ABB RobotStudio station: ABB robot domino project.rspag

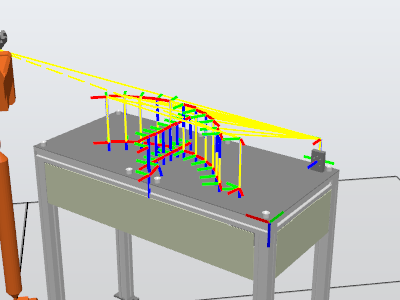
--- station ---
Station lab04_robot_mic (saved by RobotStudio 23.4.10609.1)
Controller R1400
  mechanical unit ROB_1: IRB1400_5_144__01, 6 joints, base frame (0, 0, 0) mm
Layout (positions relative to the parent item):
  - IRB1400_5_144__01 [mechanism, from Robots\IRB1400_5_144__01.rslib] at (0, 0, 0) mm; joint values [0, 0, 0, 0, 0.5236, 0] (rad or m)
  - Stoc1400 [smart component, from Components\Stoc1400.rslib] at (629.33, -613.77, 0) mm, rotated rx 0 ry 0 rz -45 deg
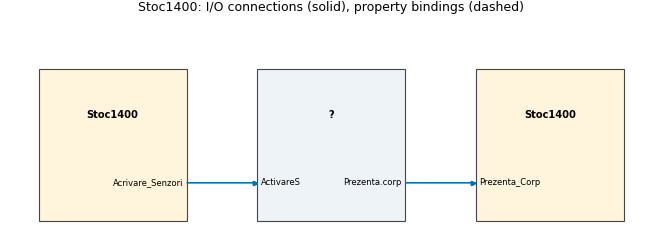
      connections:
        Stoc1400.Acrivare_Senzori -> ?.ActivareS
        Stoc1400.Acrivare_Senzori -> ?.ActivareS
        ?.Prezenta.corp -> Stoc1400.Prezenta_Corp
        ?.Prezenta.corp -> Stoc1400.Prezenta_Corp
    - 679#Body 1 [part, from Components\Stoc1400.rslib]
    - 681#Body 2 [part, from Components\Stoc1400.rslib]
    - 683#Body 3 [part, from Components\Stoc1400.rslib]
    - 685#Body 4 [part, from Components\Stoc1400.rslib]
    - 687#Body 5 [part, from Components\Stoc1400.rslib]
    - 689#Body 6 [part, from Components\Stoc1400.rslib]
    - 691#Body 7 [part, from Components\Stoc1400.rslib]
    - 693#Body 8 [part, from Components\Stoc1400.rslib]
    - 695#Body 9 [part, from Components\Stoc1400.rslib]
    - 697#Body 10 [part, from Components\Stoc1400.rslib]
    - 701#Body 12 [part, from Components\Stoc1400.rslib]
    - 703#Body 13 [part, from Components\Stoc1400.rslib]
    - 705#Body 14 [part, from Components\Stoc1400.rslib]
    - 707#Body 15 [part, from Components\Stoc1400.rslib]
    - 755#Body 39 [part, from Components\Stoc1400.rslib]
    - 757#Body 40 [part, from Components\Stoc1400.rslib]
    - 759#Body 41 [part, from Components\Stoc1400.rslib]
    - 761#Body 42 [part, from Components\Stoc1400.rslib]
    - 785#Body 54 [part, from Components\Stoc1400.rslib]
    - 787#Body 55 [part, from Components\Stoc1400.rslib]
    - 789#Body 56 [part, from Components\Stoc1400.rslib]
    - 791#Body 57 [part, from Components\Stoc1400.rslib]
    - 793#Body 58 [part, from Components\Stoc1400.rslib]
    - Part [part, from Components\Stoc1400.rslib]
    - Part_2 [part, from Components\Stoc1400.rslib]
    - Part_3 [part, from Components\Stoc1400.rslib]
    - Part_4 [part, from Components\Stoc1400.rslib]
  - Gripper_R1400 [smart component] at (943.61, 0, 1152.5) mm, rotated rx 180 ry 60 rz 180 deg
      signals: DI Open, DO Opened
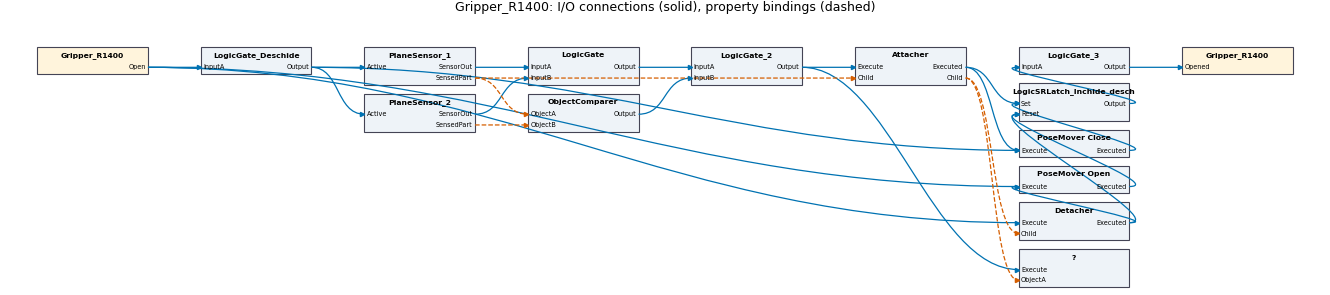
      connections:
        Attacher.Executed -> LogicSRLatch_Inchide_deschide.Set
        Detacher.Executed -> LogicSRLatch_Inchide_deschide.Reset
        Attacher.Executed -> PoseMover Close.Execute
        PoseMover Close.Executed -> LogicSRLatch_Inchide_deschide.Set
        Detacher.Executed -> PoseMover Open.Execute
        PoseMover Open.Executed -> LogicSRLatch_Inchide_deschide.Reset
        LogicGate.Output -> LogicGate_2.InputA
        ObjectComparer.Output -> LogicGate_2.InputB
        LogicGate_2.Output -> ?.Execute
        LogicGate_2.Output -> Attacher.Execute
        PlaneSensor_1.SensorOut -> LogicGate.InputA
        PlaneSensor_2.SensorOut -> LogicGate.InputB
        LogicGate_Deschide.Output -> PlaneSensor_2.Active
        LogicGate_Deschide.Output -> PlaneSensor_1.Active
        LogicGate_Deschide.Output -> PoseMover Close.Execute
        LogicSRLatch_Inchide_deschide.Output -> LogicGate_3.InputA
        LogicGate_3.Output -> Gripper_R1400.Opened
        Gripper_R1400.Open -> LogicGate_Deschide.InputA
        Gripper_R1400.Open -> Detacher.Execute
        Gripper_R1400.Open -> PoseMover Open.Execute
        Attacher.Child => Detacher.Child
        Attacher.Child => ?.ObjectA
        PlaneSensor_1.SensedPart => Attacher.Child
        PlaneSensor_1.SensedPart => ObjectComparer.ObjectA
        PlaneSensor_2.SensedPart => ObjectComparer.ObjectB
    - Attacher [smart component]
        properties: Parent=Gripper; Flange=0; Child=(none); Mount=false; Offset=[0 0 0]; Orientation=[0 0 0]
        signals: DI Execute, DO Executed
    - Detacher [smart component]
        properties: Child=(none); KeepPosition=true
        signals: DI Execute, DO Executed
    - LogicGate_Deschide [smart component]
        properties: Operator=NOT; Delay=0
        signals: DI InputA, DI InputB, DO Output
    - LogicSRLatch_Inchide_deschide [smart component]
        signals: DI Set, DI Reset, DO Output, DO InvOutput
    - PoseMover Close [smart component]
        properties: Mechanism=Gripper; Pose=3; Duration=0
        signals: DI Execute, DI Pause, DI Cancel, DO Executed, DO Executing, DO Paused
    - PoseMover Open [smart component]
        properties: Mechanism=Gripper; Pose=2; Duration=0
        signals: DI Execute, DI Pause, DI Cancel, DO Executed, DO Executing, DO Paused
    - ObjectComparer [smart component, from Components\ObjectComparer.rslib]
        properties: ObjectA=(none); ObjectB=(none)
    - LogicGate [smart component, from Components\LogicGate.rslib]
        properties: Operator=AND; Delay=0
    - LogicGate_2 [smart component, from Components\LogicGate.rslib]
        properties: Operator=AND; Delay=0
    - PlaneSensor_1 [smart component, from Components\PlaneSensor.rslib]
        properties: Origin=[-0.015 0.017 0.128]; Axis1=[2.03942606365875E-08 6.36094387840794E-09 0.0549999999999959]; Axis2=[0.03 0 0]; SensedPart=(none); Tag=(none)
      - _sensorPart_ [part], size 30 x 0 x 55 mm
    - PlaneSensor_2 [smart component, from Components\PlaneSensor.rslib]
        properties: Origin=[-0.015 -0.017 0.128]; Axis1=[0 0 0.055]; Axis2=[0.03 0 0]; SensedPart=(none); Tag=(none)
      - _sensorPart_ [part], size 30 x 0 x 55 mm
    - Gripper [mechanism] at (0, 0.03, 0) mm; joint values [0, 0] (rad or m)
        TCP Efector at (0, 0, 184.3) mm
        links: L1, L2, L3
    - LogicGate_3 [smart component, from Components\LogicGate.rslib]
        properties: Operator=NOT; Delay=0
  - Piesa_A [part, from Components\Piesa_A.rslib] at (465.74, -1014.9, 834) mm, rotated rx 84.55 ry 90 rz -140.46 deg
  - Piesa_C [part, from Components\Piesa_C.rslib] at (465.74, -1014.9, 834) mm, rotated rx 84.55 ry 90 rz -140.46 deg
  - Piesa_D [part, from Components\Piesa_D.rslib] at (465.74, -1014.9, 834) mm, rotated rx 84.55 ry 90 rz -140.46 deg
  - Piesa_C_2 [part, from Components\Piesa_C.rslib] at (465.74, -1014.9, 834) mm, rotated rx 84.55 ry 90 rz -140.46 deg
  - Piesa_C_3 [part, from Components\Piesa_C2.rslib] at (465.74, -1014.9, 834) mm, rotated rx 84.55 ry 90 rz -140.46 deg
  - Piesa_C_4 [part, from Components\Piesa_C2.rslib] at (465.74, -1014.9, 834) mm, rotated rx 84.55 ry 90 rz -140.46 deg
  - Piesa_C_5 [part, from Components\Piesa_C2.rslib] at (465.74, -1014.9, 834) mm, rotated rx 84.55 ry 90 rz -140.46 deg
  - Piesa [part, from Components\Piesa_D.rslib] at (465.74, -1014.9, 834) mm, rotated rx 84.55 ry 90 rz -140.46 deg
  - Piesa_D_2 [part, from Components\Piesa_D_1.rslib] at (465.74, -1014.9, 834) mm, rotated rx 84.55 ry 90 rz -140.46 deg
  - Piesa_E [part, from Components\Piesa_E.rslib] at (465.74, -1014.9, 834) mm, rotated rx 84.55 ry 90 rz -140.46 deg
  - Piesa_F [part, from Components\Piesa_F.rslib] at (465.74, -1014.9, 834) mm, rotated rx 84.55 ry 90 rz -140.46 deg
  - Piesa_A_2 [part, from Components\Piesa_A2.rslib] at (465.74, -1014.9, 834) mm, rotated rx 84.55 ry 90 rz -140.46 deg
  - Piesa_A_3 [part, from Components\Piesa_A3.rslib] at (465.74, -1014.9, 834) mm, rotated rx 84.55 ry 90 rz -140.46 deg
  - Piesa_A_4 [part, from Components\Piesa_A4.rslib] at (465.74, -1014.9, 834) mm, rotated rx 84.55 ry 90 rz -140.46 deg
Attachment: Gripper_R1400 is attached to IRB1400_5_144__01 / Link6
Station logic (signal -> signal, property => property):
  R1400.DO10_9 -> Gripper_R1400.Open
Targets, tools, work objects and paths stored in the station and not in the controller backup, written as RAPID:
! task T_ROB1
MODULE Module1
  CONST robtarget aPiesa:=[[50.700017393,375.465881391,-34],[0.499999623,0.499998418,-0.500001769,0.50000019],[-1,0,-1,0],[9E+09,9E+09,9E+09,9E+09,9E+09,9E+09]];
ENDMODULE


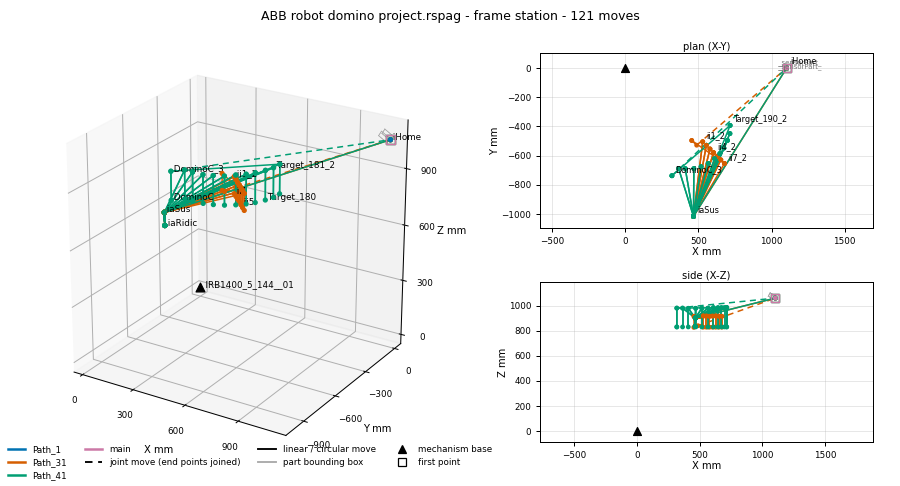
[picture p0: tool path of ABB robot domino project.rspag in frame station, 121 of 121 moves have a stored position in this frame; points joined in program order, loops and branches not executed]
--- Controller Data/R1400/RAPID/TASK1/PROGMOD/CalibData.mod ---
MODULE CalibData
ENDMODULE

--- Controller Data/R1400/RAPID/TASK1/PROGMOD/Module1.mod ---
MODULE Module1
    LOCAL PERS tooldata Efector:=[TRUE,[[0,0.033033672,184.3],[1,0,0,0]],[1.5,[0,0,90],[1,0,0,0],0.01,0.01,0.01]];
    LOCAL PERS wobjdata Paleta:=[FALSE,TRUE,"",[[164.402459193,-785.24154085,800],[0,0.923888632,0.382661463,0]],[[0,0,0],[1,0,0,0]]];
    LOCAL CONST robtarget Target_10:=[[50.700017393,375.465881391,-34],[0.69868606,0.000100025,0.000759531,-0.715427986],[0,0,0,0],[9E+09,9E+09,9E+09,9E+09,9E+09,9E+09]];
    CONST robtarget Target_20:=[[456.326,269.195,-115.604996843],[0.698683796,0.000101541,0.000757843,-0.715430199],[-1,0,-1,0],[9E+09,9E+09,9E+09,9E+09,9E+09,9E+09]];
    CONST robtarget iHome:=[[1219.122841698,108.513746508,-260.35],[0.331394548,-0.461944316,-0.191330732,-0.800111026],[0,-1,0,0],[9E+09,9E+09,9E+09,9E+09,9E+09,9E+09]];
    CONST robtarget iaSus:=[[50.700017393,375.465881391,-101.41254067],[0.707106781,0,0,-0.707106781],[-1,0,-1,0],[9E+09,9E+09,9E+09,9E+09,9E+09,9E+09]];
    CONST robtarget iaRidic:=[[52.292573517,372.97750672,-34],[0.69868606,0.000100025,0.000759531,-0.715427986],[-1,0,-1,0],[9E+09,9E+09,9E+09,9E+09,9E+09,9E+09]];
    CONST robtarget ii1_2:=[[456.326,59.195,-118.568809292],[0.698683796,0.000101541,0.000757843,-0.715430199],[0,0,0,0],[9E+09,9E+09,9E+09,9E+09,9E+09,9E+09]];
    CONST robtarget ii1:=[[456.326,59.195,-28.603],[0.698683796,0.000101541,0.000757843,-0.715430199],[0,0,0,0],[9E+09,9E+09,9E+09,9E+09,9E+09,9E+09]];
    CONST robtarget ii2_2:=[[456.326,94.195,-117.638928881],[0.698683796,0.000101541,0.000757843,-0.715430199],[0,0,0,0],[9E+09,9E+09,9E+09,9E+09,9E+09,9E+09]];
    CONST robtarget ii2:=[[456.326,94.195,-28.603],[0.698683796,0.000101541,0.000757843,-0.715430199],[0,0,0,0],[9E+09,9E+09,9E+09,9E+09,9E+09,9E+09]];
    CONST robtarget ii3_2:=[[456.326,129.195,-115.401644855],[0.698683796,0.000101541,0.000757843,-0.715430199],[0,0,0,0],[9E+09,9E+09,9E+09,9E+09,9E+09,9E+09]];
    CONST robtarget ii3:=[[456.326,129.195,-28.603],[0.698683796,0.000101541,0.000757843,-0.715430199],[0,0,0,0],[9E+09,9E+09,9E+09,9E+09,9E+09,9E+09]];
    CONST robtarget ii4_2:=[[456.326,164.195,-116.998692265],[0.698683796,0.000101541,0.000757843,-0.715430199],[0,0,0,0],[9E+09,9E+09,9E+09,9E+09,9E+09,9E+09]];
    CONST robtarget ii4:=[[456.326,164.195,-28.603],[0.698683796,0.000101541,0.000757843,-0.715430199],[0,0,0,0],[9E+09,9E+09,9E+09,9E+09,9E+09,9E+09]];
    CONST robtarget ii5_2:=[[456.326,199.195,-117.832130834],[0.698683796,0.000101541,0.000757843,-0.715430199],[0,0,0,0],[9E+09,9E+09,9E+09,9E+09,9E+09,9E+09]];
    CONST robtarget ii5:=[[456.326,199.195,-28.603],[0.698683796,0.000101541,0.000757843,-0.715430199],[0,0,0,0],[9E+09,9E+09,9E+09,9E+09,9E+09,9E+09]];
    CONST robtarget ii6_2:=[[456.326,234.195,-116.561054339],[0.698683796,0.000101541,0.000757843,-0.715430199],[0,0,0,0],[9E+09,9E+09,9E+09,9E+09,9E+09,9E+09]];
    CONST robtarget ii6:=[[456.326,234.195,-28.603],[0.698683796,0.000101541,0.000757843,-0.715430199],[0,0,0,0],[9E+09,9E+09,9E+09,9E+09,9E+09,9E+09]];
    CONST robtarget ii7_2:=[[456.326,269.195,-115.604996843],[0.698683796,0.000101541,0.000757843,-0.715430199],[0,0,0,0],[9E+09,9E+09,9E+09,9E+09,9E+09,9E+09]];
    CONST robtarget ii7:=[[456.326,269.195,-28.603],[0.698683796,0.000101541,0.000757843,-0.715430199],[0,0,0,0],[9E+09,9E+09,9E+09,9E+09,9E+09,9E+09]];
    CONST robtarget ID_Sus:=[[409.258836726,-0.15273945,-115.604996843],[0.698683796,0.000101541,0.000757843,-0.715430199],[-1,0,-1,0],[9E+09,9E+09,9E+09,9E+09,9E+09,9E+09]];
    CONST robtarget ID_Jos:=[[409.258836726,-0.15273945,-26.947996726],[0.698683796,0.000101541,0.000757843,-0.715430199],[-1,0,-1,0],[9E+09,9E+09,9E+09,9E+09,9E+09,9E+09]];
    CONST robtarget Domino:=[[410.25163548,46.685138582,-40.418213822],[0.68917084,-0.113675498,-0.121440524,-0.705247214],[-1,0,-1,0],[9E+09,9E+09,9E+09,9E+09,9E+09,9E+09]];
    CONST robtarget Target_170_2:=[[481.800724938,199.544231585,-183.999604819],[0.995072185,0,0,-0.099153148],[-1,0,0,0],[9E+09,9E+09,9E+09,9E+09,9E+09,9E+09]];
    CONST robtarget Target_170:=[[481.800724938,199.544231585,-30.630486906],[0.995072185,0,0,-0.099153148],[0,0,0,0],[9E+09,9E+09,9E+09,9E+09,9E+09,9E+09]];
    CONST robtarget Target_180_2:=[[582.438198055,172.573372066,-183.959345103],[0.97629086,0,0,-0.216462829],[-1,-1,0,0],[9E+09,9E+09,9E+09,9E+09,9E+09,9E+09]];
    CONST robtarget Target_180:=[[582.438198055,172.573372066,-30.630486906],[0.97629086,0,0,-0.216462829],[0,0,0,0],[9E+09,9E+09,9E+09,9E+09,9E+09,9E+09]];
    CONST robtarget Target_190_2:=[[667.781911679,112.809011422,-184.493963186],[0.923870432,0,0,-0.382705401],[0,0,0,0],[9E+09,9E+09,9E+09,9E+09,9E+09,9E+09]];
    CONST robtarget Target_190:=[[667.781911679,112.809011422,-30.630486906],[0.923870432,0,0,-0.382705401],[0,0,0,0],[9E+09,9E+09,9E+09,9E+09,9E+09,9E+09]];
    CONST robtarget Target_200_2:=[[306.909359491,163.530688918,-167.727227508],[0.536299591,0.000254363,0.000722629,-0.844027347],[-1,0,-1,0],[9E+09,9E+09,9E+09,9E+09,9E+09,9E+09]];
    CONST robtarget Target_200:=[[306.909359491,163.530688918,-26.975190983],[0.536299591,0.000254363,0.000722629,-0.844027347],[-1,0,-1,0],[9E+09,9E+09,9E+09,9E+09,9E+09,9E+09]];
    CONST robtarget Target_210_2:=[[354.733930359,180.209703677,-168.853762894],[0.464361971,0.000313489,0.000699011,-0.885645173],[-1,-1,-1,0],[9E+09,9E+09,9E+09,9E+09,9E+09,9E+09]];
    CONST robtarget Target_210:=[[354.733930359,180.209703677,-26.975190983],[0.464361971,0.000313489,0.000699011,-0.885645173],[-1,-1,-1,0],[9E+09,9E+09,9E+09,9E+09,9E+09,9E+09]];
    CONST robtarget Target_220_2:=[[403.502030206,179.286180207,-166.530198208],[0.375825673,0.00038013,0.000665127,-0.926690065],[-1,-1,-1,0],[9E+09,9E+09,9E+09,9E+09,9E+09,9E+09]];
    CONST robtarget Target_220:=[[403.502030206,179.286180207,-26.975190983],[0.375825673,0.00038013,0.000665127,-0.926690065],[-1,-1,-1,0],[9E+09,9E+09,9E+09,9E+09,9E+09,9E+09]];
    CONST robtarget Target_230_2:=[[451.347703104,167.719972633,-167.069743011],[0.258943654,0.000459083,0.000613298,-0.965892125],[-1,-1,-1,0],[9E+09,9E+09,9E+09,9E+09,9E+09,9E+09]];
    CONST robtarget Target_230:=[[451.347703104,167.719972633,-26.975190983],[0.258943654,0.000459083,0.000613298,-0.965892125],[-1,-1,-1,0],[9E+09,9E+09,9E+09,9E+09,9E+09,9E+09]];
    CONST robtarget DominoC_3:=[[142.859438409,74.577988932,-180.688995332],[0.393881017,0,0,-0.919161435],[-1,0,-1,0],[9E+09,9E+09,9E+09,9E+09,9E+09,9E+09]];
    CONST robtarget DominoC:=[[142.859438409,74.577988932,-30.630486906],[0.393881017,0,0,-0.919161435],[-1,0,-1,0],[9E+09,9E+09,9E+09,9E+09,9E+09,9E+09]];
    CONST robtarget Lovire:=[[241.300943539,67.077354326,-28.34493513],[0.698121404,-0.033467609,-0.042039078,-0.713960182],[-1,0,-1,0],[9E+09,9E+09,9E+09,9E+09,9E+09,9E+09]];
    CONST robtarget Target_150_2:=[[283.578545465,146.440862541,-179.015978792],[0.300007552,-0.00000002,-0.000000178,-0.953936826],[-1,-1,-1,0],[9E+09,9E+09,9E+09,9E+09,9E+09,9E+09]];
    CONST robtarget Target_160:=[[378.007856837,190.468506271,-30.630486906],[0.130502616,0,0,-0.991447965],[-1,-1,-1,0],[9E+09,9E+09,9E+09,9E+09,9E+09,9E+09]];
    CONST robtarget Target_171_2:=[[528.22113049,192.308253683,-184.191222664],[0.984830453,0,0,-0.173519391],[-1,-1,0,0],[9E+09,9E+09,9E+09,9E+09,9E+09,9E+09]];
    CONST robtarget Target_171:=[[528.22113049,192.308253683,-30.630486906],[0.984830453,0,0,-0.173519391],[-1,-1,0,0],[9E+09,9E+09,9E+09,9E+09,9E+09,9E+09]];
    CONST robtarget Target_141:=[[241.884072512,104.750355256,-30.630486906],[0.349991593,0,0,-0.936752841],[-1,0,-1,0],[9E+09,9E+09,9E+09,9E+09,9E+09,9E+09]];
    CONST robtarget Target_140:=[[209.902359402,72.771684008,-30.562172725],[0.393881017,0,0,-0.919161435],[-1,0,-1,0],[9E+09,9E+09,9E+09,9E+09,9E+09,9E+09]];
    CONST robtarget Target_140_2:=[[209.902359402,72.771684008,-180.562172725],[0.393881017,0,0,-0.919161435],[-1,0,-1,0],[9E+09,9E+09,9E+09,9E+09,9E+09,9E+09]];
    CONST robtarget Target_150:=[[283.616805576,146.386732955,-30.630438676],[0.300007552,-0.00000002,-0.000000178,-0.953936826],[-1,-1,-1,0],[9E+09,9E+09,9E+09,9E+09,9E+09,9E+09]];
    CONST robtarget Target_161_2:=[[431.263927092,198.857293079,-184.181538316],[0.021799568,0,0,-0.999762361],[-1,-1,-1,0],[9E+09,9E+09,9E+09,9E+09,9E+09,9E+09]];
    CONST robtarget Target_141_2:=[[241.884072512,104.750355256,-179.064848292],[0.349991593,0,0,-0.936752841],[-1,0,-1,0],[9E+09,9E+09,9E+09,9E+09,9E+09,9E+09]];
    CONST robtarget Target_151_2:=[[327.822781481,171.759911975,-180.139566205],[0.223808464,0,0,-0.974633147],[-1,0,-1,0],[9E+09,9E+09,9E+09,9E+09,9E+09,9E+09]];
    CONST robtarget Target_181:=[[627.363553937,151.187326706,-30.978234387],[0.949049924,0,0,-0.315125754],[-1,-1,0,0],[9E+09,9E+09,9E+09,9E+09,9E+09,9E+09]];
    CONST robtarget Target_151:=[[327.822781481,171.759911975,-30.630486906],[0.223808464,0,0,-0.974633147],[-1,-1,-1,0],[9E+09,9E+09,9E+09,9E+09,9E+09,9E+09]];
    CONST robtarget Target_161:=[[431.263927092,198.857293079,-30.630486906],[0.021799568,0,0,-0.999762361],[-1,-1,-1,0],[9E+09,9E+09,9E+09,9E+09,9E+09,9E+09]];
    CONST robtarget Target_160_2:=[[378.007856837,190.468506271,-180.335566752],[0.130502616,0,0,-0.991447965],[-1,-1,-1,0],[9E+09,9E+09,9E+09,9E+09,9E+09,9E+09]];
    CONST robtarget Target_181_2:=[[627.363553937,151.187326706,-184.978843448],[0.949049924,0,0,-0.315125754],[-1,-1,0,0],[9E+09,9E+09,9E+09,9E+09,9E+09,9E+09]];
    CONST robtarget LovireCerc:=[[142.868157241,74.605504654,-30.630477518],[0.756533746,0.000000012,0.000000022,-0.653954656],[-1,0,-1,0],[9E+09,9E+09,9E+09,9E+09,9E+09,9E+09]];
    LOCAL PROC Path_1()
        MoveJ iHome,v300,fine,Efector\WObj:=Paleta;
    ENDPROC

    LOCAL PROC Path_31()
        Set DO10_9;
        WaitTime 0.5;
        MoveJ iHome,v300,fine,Efector\WObj:=Paleta;
        WaitTime 0.5;
        MoveL iaSus,v300,fine,Efector\WObj:=Paleta;
        WaitTime 0.5;
        MoveL iaRidic,v300,fine,Efector\WObj:=Paleta;
        WaitTime 0.5;
        Reset DO10_9;
        WaitTime 0.5;
        MoveL iaSus,v300,fine,Efector\WObj:=Paleta;
        WaitTime 0.5;
        MoveL ii1_2,v300,fine,Efector\WObj:=Paleta;
        WaitTime 0.5;
        MoveL ii1,v300,fine,Efector\WObj:=Paleta;
        Set DO10_9;
        WaitTime 0.5;
        MoveL ii1_2,v300,fine,Efector\WObj:=Paleta;
        WaitTime 0.5;
        MoveL iaSus,v300,fine,Efector\WObj:=Paleta;
        WaitTime 0.5;
        MoveL iaRidic,v300,fine,Efector\WObj:=Paleta;
        WaitTime 0.5;
        Reset DO10_9;
        WaitTime 0.5;
        MoveL iaSus,v300,fine,Efector\WObj:=Paleta;
        WaitTime 0.5;
        Reset DO10_9;
        WaitTime 0.5;
        MoveL ii2_2,v300,fine,Efector\WObj:=Paleta;
        WaitTime 0.5;
        MoveL ii2,v300,fine,Efector\WObj:=Paleta;
        WaitTime 0.5;
        Set DO10_9;
        WaitTime 0.5;
        MoveL ii2_2,v300,fine,Efector\WObj:=Paleta;
        WaitTime 0.5;
        MoveL iaSus,v300,fine,Efector\WObj:=Paleta;
        WaitTime 0.5;
        MoveL iaRidic,v300,fine,Efector\WObj:=Paleta;
        WaitTime 0.5;
        Reset DO10_9;
        WaitTime 0.5;
        MoveL iaSus,v300,fine,Efector\WObj:=Paleta;
        WaitTime 0.5;
        Reset DO10_9;
        WaitTime 0.5;
        MoveL ii3_2,v300,fine,Efector\WObj:=Paleta;
        WaitTime 0.5;
        MoveL ii3,v300,fine,Efector\WObj:=Paleta;
        WaitTime 0.5;
        Set DO10_9;
        WaitTime 0.5;
        MoveL ii3_2,v300,fine,Efector\WObj:=Paleta;
        WaitTime 0.5;
        MoveL iaSus,v300,fine,Efector\WObj:=Paleta;
        WaitTime 0.5;
        MoveL iaRidic,v300,fine,Efector\WObj:=Paleta;
        WaitTime 0.5;
        Reset DO10_9;
        WaitTime 0.5;
        MoveL iaSus,v300,fine,Efector\WObj:=Paleta;
        WaitTime 0.5;
        Reset DO10_9;
        WaitTime 0.5;
        MoveL ii4_2,v300,fine,Efector\WObj:=Paleta;
        WaitTime 0.5;
        MoveL ii4,v300,fine,Efector\WObj:=Paleta;
        WaitTime 0.5;
        Set DO10_9;
        WaitTime 0.5;
        MoveL ii4_2,v300,fine,Efector\WObj:=Paleta;
        WaitTime 0.5;
        MoveL iaSus,v300,fine,Efector\WObj:=Paleta;
        WaitTime 0.5;
        MoveL iaRidic,v300,fine,Efector\WObj:=Paleta;
        WaitTime 0.5;
        Reset DO10_9;
        MoveL iaSus,v300,fine,Efector\WObj:=Paleta;
        WaitTime 0.5;
        Reset DO10_9;
        WaitTime 0.5;
        MoveL ii5_2,v300,fine,Efector\WObj:=Paleta;
        WaitTime 0.5;
        MoveL ii5,v300,fine,Efector\WObj:=Paleta;
        WaitTime 0.5;
        Set DO10_9;
        WaitTime 0.5;
        MoveL ii5_2,v300,fine,Efector\WObj:=Paleta;
        WaitTime 0.5;
        MoveL iaSus,v300,fine,Efector\WObj:=Paleta;
        WaitTime 0.5;
        MoveL iaRidic,v300,fine,Efector\WObj:=Paleta;
        WaitTime 0.5;
        Reset DO10_9;
        MoveL iaSus,v300,fine,Efector\WObj:=Paleta;
        WaitTime 0.5;
        Reset DO10_9;
        WaitTime 0.5;
        MoveL ii6_2,v300,fine,Efector\WObj:=Paleta;
        WaitTime 0.5;
        MoveL ii6,v300,fine,Efector\WObj:=Paleta;
        WaitTime 0.5;
        Set DO10_9;
        WaitTime 0.5;
        MoveL ii6_2,v300,fine,Efector\WObj:=Paleta;
        WaitTime 0.5;
        MoveL iaSus,v300,fine,Efector\WObj:=Paleta;
        WaitTime 0.5;
        MoveL iaRidic,v300,fine,Efector\WObj:=Paleta;
        WaitTime 0.5;
        WaitTime 0.5;
        Reset DO10_9;
        WaitTime 0.5;
        MoveL iaSus,v300,fine,Efector\WObj:=Paleta;
        WaitTime 0.5;
        Reset DO10_9;
        WaitTime 0.5;
        MoveL ii7_2,v300,fine,Efector\WObj:=Paleta;
        WaitTime 0.5;
        MoveL ii7,v300,fine,Efector\WObj:=Paleta;
        WaitTime 0.5;
        Set DO10_9;
        WaitTime 0.5;
        MoveL ii7_2,v300,fine,Efector\WObj:=Paleta;
        WaitTime 0.5;
        Set DO10_9;
        WaitTime 0.5;
        MoveL ID_Sus,v300,fine,Efector\WObj:=Paleta;
        WaitTime 0.5;
        MoveL ID_Jos,v300,fine,Efector\WObj:=Paleta;
        WaitTime 0.5;
        MoveL Domino,v300,fine,Efector\WObj:=Paleta;
        WaitTime 0.5;
        MoveJ iHome,v300,fine,Efector\WObj:=Paleta;
    ENDPROC

    PROC Path_41()
        Set DO10_9;
        WaitTime 0.5;
        MoveJ iHome,v300,fine,Efector\WObj:=Paleta;
        WaitTime 0.5;
        MoveL iaSus,v300,fine,Efector\WObj:=Paleta;
        WaitTime 0.5;
        MoveL iaRidic,v300,fine,Efector\WObj:=Paleta;
        WaitTime 0.5;
        Reset DO10_9;
        WaitTime 0.5;
        MoveL iaSus,v300,fine,Efector\WObj:=Paleta;
        WaitTime 0.5;
        MoveL Target_140_2,v300,fine,Efector\WObj:=Paleta;
        MoveL Target_140,v300,fine,Efector\WObj:=Paleta;
        WaitTime 0.5;
        Set DO10_9;
        WaitTime 0.5;
        MoveL Target_140_2,v300,fine,Efector\WObj:=Paleta;
        MoveL iaSus,v300,fine,Efector\WObj:=Paleta;
        WaitTime 0.5;
        MoveL iaRidic,v300,fine,Efector\WObj:=Paleta;
        WaitTime 0.5;
        Reset DO10_9;
        WaitTime 0.5;
        MoveL iaSus,v300,fine,Efector\WObj:=Paleta;
        WaitTime 0.5;
        MoveL Target_141_2,v300,fine,Efector\WObj:=Paleta;
        MoveL Target_141,v300,fine,Efector\WObj:=Paleta;
        WaitTime 0.5;
        Set DO10_9;
        WaitTime 0.5;
        MoveL Target_141_2,v300,fine,Efector\WObj:=Paleta;
        MoveL iaSus,v300,fine,Efector\WObj:=Paleta;
        WaitTime 0.5;
        MoveL iaRidic,v300,fine,Efector\WObj:=Paleta;
        WaitTime 0.5;
        Reset DO10_9;
        WaitTime 0.5;
        MoveL iaSus,v300,fine,Efector\WObj:=Paleta;
        WaitTime 0.5;
        MoveL Target_150_2,v300,fine,Efector\WObj:=Paleta;
        MoveL Target_150,v300,fine,Efector\WObj:=Paleta;
        WaitTime 0.5;
        Set DO10_9;
        WaitTime 0.5;
        MoveL Target_150_2,v300,fine,Efector\WObj:=Paleta;
        MoveL iaSus,v300,fine,Efector\WObj:=Paleta;
        WaitTime 0.5;
        MoveL iaRidic,v300,fine,Efector\WObj:=Paleta;
        WaitTime 0.5;
        Reset DO10_9;
        WaitTime 0.5;
        MoveL iaSus,v300,fine,Efector\WObj:=Paleta;
        WaitTime 0.5;
        MoveL Target_151_2,v300,fine,Efector\WObj:=Paleta;
        MoveL Target_151,v300,fine,Efector\WObj:=Paleta;
        WaitTime 0.5;
        Set DO10_9;
        WaitTime 0.5;
        MoveL Target_151_2,v300,fine,Efector\WObj:=Paleta;
        MoveL iaSus,v300,fine,Efector\WObj:=Paleta;
        WaitTime 0.5;
        MoveL iaRidic,v300,fine,Efector\WObj:=Paleta;
        WaitTime 0.5;
        Reset DO10_9;
        WaitTime 0.5;
        MoveL iaSus,v300,fine,Efector\WObj:=Paleta;
        WaitTime 0.5;
        MoveL Target_160_2,v300,fine,Efector\WObj:=Paleta;
        MoveL Target_160,v300,fine,Efector\WObj:=Paleta;
        WaitTime 0.5;
        Set DO10_9;
        WaitTime 0.5;
        MoveL Target_160_2,v300,fine,Efector\WObj:=Paleta;
        MoveL iaSus,v300,fine,Efector\WObj:=Paleta;
        WaitTime 0.5;
        MoveL iaRidic,v300,fine,Efector\WObj:=Paleta;
        WaitTime 0.5;
        Reset DO10_9;
        WaitTime 0.5;
        MoveL iaSus,v300,fine,Efector\WObj:=Paleta;
        WaitTime 0.5;
        MoveL Target_161_2,v300,fine,Efector\WObj:=Paleta;
        MoveL Target_161,v300,fine,Efector\WObj:=Paleta;
        WaitTime 0.5;
        Set DO10_9;
        WaitTime 0.5;
        MoveL Target_161_2,v300,fine,Efector\WObj:=Paleta;
        MoveL iaSus,v300,fine,Efector\WObj:=Paleta;
        WaitTime 0.5;
        MoveL iaRidic,v300,fine,Efector\WObj:=Paleta;
        WaitTime 0.5;
        Reset DO10_9;
        WaitTime 0.5;
        MoveL iaSus,v300,fine,Efector\WObj:=Paleta;
        WaitTime 0.5;
        MoveL Target_170_2,v300,fine,Efector\WObj:=Paleta;
        MoveL Target_170,v300,fine,Efector\WObj:=Paleta;
        WaitTime 0.5;
        Set DO10_9;
        WaitTime 0.5;
        MoveL Target_170_2,v300,fine,Efector\WObj:=Paleta;
        MoveL iaSus,v300,fine,Efector\WObj:=Paleta;
        WaitTime 0.5;
        MoveL iaRidic,v300,fine,Efector\WObj:=Paleta;
        WaitTime 0.5;
        Reset DO10_9;
        WaitTime 0.5;
        MoveL iaSus,v300,fine,Efector\WObj:=Paleta;
        WaitTime 0.5;
        MoveL Target_171_2,v300,fine,Efector\WObj:=Paleta;
        MoveL Target_171,v300,fine,Efector\WObj:=Paleta;
        WaitTime 0.5;
        Set DO10_9;
        WaitTime 0.5;
        MoveL Target_171_2,v300,fine,Efector\WObj:=Paleta;
        MoveL iaSus,v300,fine,Efector\WObj:=Paleta;
        WaitTime 0.5;
        MoveL iaRidic,v300,fine,Efector\WObj:=Paleta;
        WaitTime 0.5;
        Reset DO10_9;
        WaitTime 0.5;
        MoveL iaSus,v300,fine,Efector\WObj:=Paleta;
        WaitTime 0.5;
        MoveL Target_180_2,v300,fine,Efector\WObj:=Paleta;
        MoveL Target_180,v300,fine,Efector\WObj:=Paleta;
        WaitTime 0.5;
        Set DO10_9;
        WaitTime 0.5;
        MoveL Target_180_2,v300,fine,Efector\WObj:=Paleta;
        MoveL iaSus,v300,fine,Efector\WObj:=Paleta;
        WaitTime 0.5;
        MoveL iaRidic,v300,fine,Efector\WObj:=Paleta;
        WaitTime 0.5;
        Reset DO10_9;
        WaitTime 0.5;
        MoveL iaSus,v300,fine,Efector\WObj:=Paleta;
        WaitTime 0.5;
        MoveL Target_181_2,v300,fine,Efector\WObj:=Paleta;
        MoveL Target_181,v300,fine,Efector\WObj:=Paleta;
        WaitTime 0.5;
        Set DO10_9;
        WaitTime 0.5;
        MoveL Target_181_2,v300,fine,Efector\WObj:=Paleta;
        MoveL iaSus,v300,fine,Efector\WObj:=Paleta;
        WaitTime 0.5;
        MoveL iaRidic,v300,fine,Efector\WObj:=Paleta;
        WaitTime 0.5;
        Reset DO10_9;
        WaitTime 0.5;
        MoveL iaSus,v300,fine,Efector\WObj:=Paleta;
        WaitTime 0.5;
        MoveL Target_190_2,v300,fine,Efector\WObj:=Paleta;
        MoveL Target_190,v300,fine,Efector\WObj:=Paleta;
        WaitTime 0.5;
        Set DO10_9;
        WaitTime 0.5;
        MoveL Target_190_2,v300,fine,Efector\WObj:=Paleta;
        WaitTime 0.5;
        MoveL DominoC_3,v300,fine,Efector\WObj:=Paleta;
        WaitTime 0.5;
        MoveL DominoC,v300,fine,Efector\WObj:=Paleta;
        WaitTime 0.5;
        MoveL LovireCerc,v300,fine,Efector\WObj:=Paleta;
        WaitTime 0.5;
        MoveL DominoC_3,v300,fine,Efector\WObj:=Paleta;
        WaitTime 0.5;
        MoveJ iHome,v300,fine,Efector\WObj:=Paleta;
    ENDPROC

   PROC TargetHome(robtarget t1)
       VAR num x1;
       VAR num x2;
       VAR num x3;
       VAR num x4;
       x1:=t1.robconf.cf1;
       x2:=t1.robconf.cf4;
       x3:=t1.robconf.cf6;
       x4:=t1.robconf.cfx;
       TPWrite "Configuratie targetului HOME este:";
       TPWrite "Configuratia cf1="\Num:=x1;
       TPWrite "Configuratia cf4="\Num:=x2;
       TPWrite "Configuratia cf6="\Num:=x3;
       TPWrite "Configuratia cfx="\Num:=x4;
   ENDPROC

    FUNC bool Pozitionare(robtarget t1, robtarget t2)
        VAR num x1;
        VAR num x2;
        x1:=t1.trans.x;
        x2:=t2.trans.x;
        IF x1=x2 THEN
            TPWrite "Valoarea de pozitionare ESTE egala pentru cele 2 targeturi!";
            RETURN TRUE;
        ELSE
            TPWrite "Valoarea de pozitionare NU este egala pentru cele 2 targeturi!";
            RETURN FALSE;
        ENDIF
    ENDFUNC
    PROC main()
            VAR num cerere;
            VAR num valoare;
            VAR num calcul;
            VAR bool egal;
            TPReadFK cerere,"Ce sa construiesc?","Linie","Cerc","Nimic?",stEmpty,stEmpty;
            IF cerere=1 THEN
                TPWrite "S-a selectat linia";
                Path_31;
            ELSEIF cerere=2 THEN
                TPWrite "S-a selectat arcul de cerc";
                Path_41;
            ELSEIF cerere=3 THEN
                TPWrite "S-a selectat nimic, deci merg acasa...";
                MoveJ iHome,v300,fine,Efector\WObj:=Paleta;
                TPReadNum calcul,"Vrei sa afisez date despre targetul iHome?  1-Config / 2-Pozitie / 3-NU";
                IF calcul=1 THEN
                    TargetHome(iHome);
                ELSEIF calcul=2 THEN
                    TPWrite "Afisez daca iHome si DominoC au aceeasi pozitie pe x: ";
                    egal:=Pozitionare(iHome,DominoC);
                ELSEIF calcul=3 THEN
                    TPWrite "Finalizare task!";
                ENDIF
            ENDIF
    ENDPROC



ENDMODULE

--- Controller Data/R1400/SYSPAR/EIO.cfg ---
EIO:CFG_1.0:5:60::
#
EIO_BUS:

      -Name "Virtual1"
#
EIO_UNIT_TYPE:

      -Name "Virtual" -VendorName "ABB" -ProductName "Virtual unit"
#
EIO_UNIT:

      -Name "TuIasi" -UnitType "Virtual" -Bus "Virtual1"
#
EIO_SIGNAL:

      -Name "DO10_9" -SignalType "DO" -Unit "TuIasi" -UnitMap "1" -Access "All"

      -Name "DO11_7" -SignalType "DO" -Unit "TuIasi" -UnitMap "2" -Access "All"

      -Name "DO11_8" -SignalType "DO" -Unit "TuIasi" -UnitMap "3" -Access "All"

      -Name "DO11_9" -SignalType "DO" -Unit "TuIasi" -UnitMap "4" -Access "All"

      -Name "DO12_1" -SignalType "DO" -Unit "TuIasi" -UnitMap "5" -Access "All"

      -Name "DO13_1" -SignalType "DO" -Unit "TuIasi" -UnitMap "7" -Access "All"

      -Name "DI11_9" -SignalType "DI" -Unit "TuIasi" -UnitMap "8" -Access "All"

      -Name "DI13_9" -SignalType "DI" -Unit "TuIasi" -UnitMap "9" -Access "All"

      -Name "AO12_1" -SignalType "AO" -Unit "TuIasi" -UnitMap "16-31"\
      -Access "All"

      -Name "DI12_2" -SignalType "DI" -Unit "TuIasi" -UnitMap "10" -Access "All"

      -Name "DO12_10" -SignalType "DO" -Unit "TuIasi" -UnitMap "11"\
      -Access "All"

      -Name "DI10_1" -SignalType "DI" -Unit "TuIasi" -UnitMap "12" -Access "All"

      -Name "DI10_7" -SignalType "DI" -Unit "TuIasi" -UnitMap "13" -Access "All"

      -Name "DI10_6" -SignalType "DI" -Unit "TuIasi" -UnitMap "14" -Access "All"

      -Name "DI10_5" -SignalType "DI" -Unit "TuIasi" -UnitMap "15" -Access "All"

      -Name "DI10_4" -SignalType "DI" -Unit "TuIasi" -UnitMap "32" -Access "All"

      -Name "DO10_3" -SignalType "DO" -Unit "TuIasi" -UnitMap "33" -Access "All"

      -Name "DO10_4" -SignalType "DO" -Unit "TuIasi" -UnitMap "34" -Access "All"

      -Name "DO10_2" -SignalType "DO" -Unit "TuIasi" -UnitMap "35" -Access "All"

      -Name "DO10_1" -SignalType "DO" -Unit "TuIasi" -UnitMap "36" -Access "All"
#
EIO_ACCESS:

      -Name "All" -Rapid  -LocalManual  -LocalAuto  -RemoteManual  -RemoteAuto
